// TwinCAT 3 PLC project Bridge
// ProgramVersion: 3.1.4023.0
// libraries:
//   Tc2_Standard, * (Beckhoff Automation GmbH)
//   Tc2_System, * (Beckhoff Automation GmbH)
//   Tc3_Module, * (Beckhoff Automation GmbH)
// project tree:
//   / Class Diagram.TcCD (not stored), PlcTask.TcTTO
//   Classes/ FB_Shape.TcPOU, FB_RedColor.TcPOU, FB_BlueColor.TcPOU, FB_Square.TcPOU, FB_Circle.TcPOU
//   Interfaces/ ITF_Color.TcIO
//   POUs/ MAIN.TcPOU
// real-time tasks:
//   TASK PlcTask: cycle T#10ms, priority 20, ADS port 350

CONFIGURATION Bridge
    RESOURCE PLC ON TwinCAT3
        TASK PlcTask(INTERVAL := T#10ms, PRIORITY := 20);
        PROGRAM MAIN WITH PlcTask : MAIN;
    END_RESOURCE
END_CONFIGURATION

// ---- Interfaces/ITF_Color.TcIO
INTERFACE ITF_Color

METHOD applyColor : STRING
END_METHOD

END_INTERFACE

// ---- POUs/MAIN.TcPOU
PROGRAM MAIN
VAR
	
     fbRedColor 		: FB_RedColor;
	 fbBlueColor 		: FB_BlueColor;
	 
	 fbSquareRed 		: FB_Square(Color:= fbRedColor );
	 fbSquareBlue 		: FB_Square(Color:= fbBlueColor );
	 
	 fbCircleRed 		: FB_Circle(Color:= fbRedColor );
	 fbCircleBlue 		: FB_Circle(Color:= fbBlueColor );
	 
	 bstartDemo1		: BOOL;
	 
END_VAR

IF bstartDemo1 THEN
	bstartDemo1 := FALSE;
	
	fbSquareRed.Draw();
	fbSquareBlue.Draw();
	
	fbCircleRed.Draw();
	fbCircleBlue.Draw();
	
END_IF

END_PROGRAM

// ---- Classes/FB_RedColor.TcPOU
FUNCTION_BLOCK FB_RedColor IMPLEMENTS ITF_Color

METHOD applyColor : STRING
applyColor := 'red';
END_METHOD

END_FUNCTION_BLOCK

// ---- Classes/FB_BlueColor.TcPOU
FUNCTION_BLOCK FB_BlueColor IMPLEMENTS ITF_Color

METHOD applyColor : STRING
applyColor := 'blue';
END_METHOD

END_FUNCTION_BLOCK

// ---- Classes/FB_Square.TcPOU
FUNCTION_BLOCK FB_Square EXTENDS FB_Shape

METHOD Draw : STRING
ADSLOGSTR(    msgCtrlMask:=ADSLOG_MSGTYPE_LOG,
              msgFmtStr:='Drawing a %s square',
              strArg:= SUPER^._color.applyColor());
END_METHOD

END_FUNCTION_BLOCK

// ---- Classes/FB_Shape.TcPOU
FUNCTION_BLOCK ABSTRACT FB_Shape
VAR
	_color : ITF_color;
END_VAR

METHOD ABSTRACT Draw : STRING
END_METHOD

METHOD FB_init : BOOL
VAR_INPUT
	bInitRetains : BOOL; // if TRUE, the retain variables are initialized (warm start / cold start)
	bInCopyCode : BOOL;  // if TRUE, the instance afterwards gets moved into the copy code (online change)
	Color : ITF_Color;
END_VAR
THIS^._color := Color;
END_METHOD

END_FUNCTION_BLOCK

// ---- Classes/FB_Circle.TcPOU
FUNCTION_BLOCK FB_Circle EXTENDS FB_Shape

METHOD Draw : STRING
ADSLOGSTR(    msgCtrlMask:=ADSLOG_MSGTYPE_LOG,
              msgFmtStr:='Drawing a %s circle',
              strArg:= SUPER^._color.applyColor());
END_METHOD

END_FUNCTION_BLOCK
